{attribute 'linkalways'} 
{attribute 'no_explicit_call' := 'This FB is a CLASS and must be accessed using methods or properties'}
{attribute 'enable_dynamic_creation'}
FUNCTION_BLOCK ABSTRACT ArrayDatatypeBase_1D EXTENDS UserDefinedDatatypeBase IMPLEMENTS I_ArrayDatatype_1D
VAR
END_VAR

PROPERTY PUBLIC ABSTRACT BaseDatatype : I_Datatype
GET
END_GET
END_PROPERTY

PROPERTY Dimention : UDINT
GET
Dimention := 1;
END_GET
END_PROPERTY

PROPERTY PUBLIC Identifier : T_MAXSTRING
GET
VAR
	baseTypeAsUdt : I_UserDefinedDatatype;
	lowerBound : DINT;
	upperBound : DINT;
END_VAR
TryGetLowerBound(1, lowerBound);
TryGetUpperBound(1, upperBound);

Identifier := Concat('ARRAY [', DINT_TO_STRING(lowerBound));
Identifier := Concat(Identifier,'..');
Identifier := Concat(Identifier, DINT_TO_STRING(upperBound));
Identifier := Concat(Identifier, '] OF ');

IF BaseDatatype.TryResolveAsUserDefinedDatatype(baseTypeAsUdt) THEN
	Identifier := Concat(Identifier, baseTypeAsUdt.Identifier);
ELSE
	Identifier := Concat(Identifier, BaseDatatype.TypeName);
END_IF
END_GET
END_PROPERTY

PROPERTY PUBLIC Length : UDINT
GET
VAR
	lowerBound : DINT;
	upperBound : DINT;
END_VAR
TryGetLowerBound(1, lowerBound);
TryGetUpperBound(1, upperBound);
Length := DINT_TO_UDINT(ABS(upperBound - lowerBound) + 1);
END_GET
END_PROPERTY

METHOD PROTECTED ABSTRACT OnSerializeArrayValues
VAR_INPUT
	Serializer : I_Serializer;
END_VAR
END_METHOD

METHOD PROTECTED OnSerializeTypeWith
VAR_INPUT
	Serializer : I_Serializer;
END_VAR
SUPER^.OnSerializeTypeWith(Serializer);
SerializeBaseType(Serializer);
END_METHOD

METHOD PRIVATE SerializeBaseType
VAR_INPUT
	Serializer : I_Serializer;
END_VAR
IF BaseDatatype = 0 THEN
	RETURN;
END_IF

Serializer.AddKey('baseType');
BaseDatatype.SerializeTypeWith(Serializer);
END_METHOD

METHOD PUBLIC SerializeWith
VAR_INPUT
	Serializer : I_Serializer;
END_VAR
Serializer.StartArray();
OnSerializeArrayValues(Serializer);
Serializer.EndArray();
END_METHOD

METHOD PROTECTED ABSTRACT TryDeserializeArrayValues : BOOL
VAR_INPUT
	Deserializer : I_Deserializer;
	Feedback : I_DeserializerFeedback;
END_VAR
END_METHOD

METHOD TryDeserializeFrom : BOOL
VAR_INPUT
	Deserializer : I_Deserializer;
	Feedback : I_DeserializerFeedback;
END_VAR
TryDeserializeFrom := TryDeserializeArrayValues(Deserializer, Feedback);
END_METHOD

METHOD PUBLIC ABSTRACT TryGetElementAsDatatypeByIndex : BOOL
VAR_INPUT
	Index : DINT;
	Destination : REFERENCE TO I_Datatype;
END_VAR
END_METHOD

METHOD PUBLIC ABSTRACT TryGetLowerBound : BOOL
VAR_INPUT
	Dimention : UDINT;
	Destination : REFERENCE TO DINT;
END_VAR
END_METHOD

METHOD PUBLIC ABSTRACT TryGetUpperBound : BOOL
VAR_INPUT
	Dimention : UDINT;
	Destination : REFERENCE TO DINT;
END_VAR
END_METHOD

METHOD PUBLIC TryResolveAs1DArrayDatatype : BOOL
VAR_INPUT
	Destination : REFERENCE TO I_ArrayDatatype_1D;
END_VAR
Destination := THIS^;
TryResolveAs1DArrayDatatype := TRUE;
END_METHOD

METHOD PUBLIC TryResolveAs2DArrayDatatype : BOOL
VAR_INPUT
	Destination : REFERENCE TO I_ArrayDatatype_2D;
END_VAR
TryResolveAs2DArrayDatatype := FALSE;
END_METHOD

METHOD PUBLIC TryResolveAs3DArrayDatatype : BOOL
VAR_INPUT
	Destination : REFERENCE TO I_ArrayDatatype_3D;
END_VAR
TryResolveAs3DArrayDatatype := FALSE;
END_METHOD

METHOD PUBLIC TryResolveAsArrayDatatype : BOOL
VAR_INPUT
	Destination : REFERENCE TO I_ArrayDatatype;
END_VAR
Destination := THIS^;
TryResolveAsArrayDatatype := TRUE;
END_METHOD

PROPERTY PUBLIC TypeName : T_MAXSTRING
GET
TypeName := 'ARRAY';
END_GET
END_PROPERTY

END_FUNCTION_BLOCK

(* stored: Version 1.1.0.1, ProductVersion 3.1.4024.13
   POU ArrayDatatypeBase_1D: Id {991b8878-a517-02d7-2a23-e8a5c4d992bd}, SpecialFunc None
   Folder Private: Id {a0b3f2c8-538b-0d38-2337-b28ef79dc85d}
   Folder Protected: Id {63cbfb38-749c-0fb5-2a44-a437ca7a7a1f}
   Property BaseDatatype: Id {e7cc5988-3f2b-0d88-33df-f9d96da8e186}
   Get Get: Id {d831321b-2565-0f88-0f30-441c93e1dfda}
   Property Dimention: Id {799784aa-360e-020e-0d78-26bc6f329485}
   Get Get: Id {74727b2e-4a13-0724-3e64-b9a21a3f9986}
   Property Identifier: Id {2fb82553-7435-463b-94b6-edc871a50638}
   Get Get: Id {3f40e6ca-bcce-4ae5-ab8f-039359f2d5b2}
   Property Length: Id {c8df4437-652c-04b8-35c6-4856f897a24a}
   Get Get: Id {a600413a-c09c-0e5c-1f92-3e6a4da4c8af}
   Method OnSerializeArrayValues: Id {9b19600a-3aab-0e34-2593-3ab26ca49a5c}
   Method OnSerializeTypeWith: Id {1912559b-ea52-07bd-3eb2-f36f75f918bc}
   Method SerializeBaseType: Id {17ec54ac-5ca8-0857-3bd8-63d2ae8f5f0d}
   Method SerializeWith: Id {684d239f-36a7-0f60-36e3-867125d46b0d}
   Method TryDeserializeArrayValues: Id {c71a1318-b78e-07d7-099f-0801c70cb09d}
   Method TryDeserializeFrom: Id {02cc8c70-2927-0c70-1010-8e0f185e7fac}
   Method TryGetElementAsDatatypeByIndex: Id {72faebb8-2123-0fbb-3cbb-f1f40ed95eb1}
   Method TryGetLowerBound: Id {38b1a3d6-2dac-0ca3-32e5-50b5463b422b}
   Method TryGetUpperBound: Id {e2fa2c9f-20a5-0726-208b-61f7911bf99d}
   Method TryResolveAs1DArrayDatatype: Id {5dd922ee-79e6-0c9a-0e6b-27056823af4a}
   Method TryResolveAs2DArrayDatatype: Id {d0feb899-7b23-0e83-03c9-08c54f61fec7}
   Method TryResolveAs3DArrayDatatype: Id {224deabd-d543-06f0-2439-f7ca355ff8e2}
   Method TryResolveAsArrayDatatype: Id {36f0ff38-3d27-0156-1669-e3996fafb148}
   Property TypeName: Id {51bf05b3-954f-0c7d-072e-7f4beab269b3}
   Get Get: Id {3101e7aa-7e80-06b0-0ff0-1ad591f00d35} *)
